// TIA Portal V18 export
FUNCTION "FC_Teach_Recipe_Transfer" : Void   // FC4, SCL
{ S7_Optimized_Access := 'TRUE' }
// stored: SetENOAutomatically false
   VAR_IN_OUT
      recipeIndex : USInt;
   END_VAR
BEGIN

   // Clamp recipe index to array bounds [1..10].
   // 
   IF #recipeIndex< 1 THEN
     #recipeIndex := 1;
   ELSIF #recipeIndex> 10 THEN
     #recipeIndex := 10;
   END_IF;

   // Block read/save if teach mode is not active.
   IF NOT "DB_PARAMETERS_TEACH".HMI_PAGE_CONTROL.TEACH_MODE_ACTIVE THEN
     "DB_PARAMETERS_TEACH".HMI_PAGE_CONTROL.READ_CHOOSED_RECIPE := FALSE;
     "DB_PARAMETERS_TEACH".HMI_PAGE_CONTROL.SAVE_CHANGES_IN_RECIPE := FALSE;
     RETURN;
   END_IF;

   // Read selected recipe into teach screen values.
   IF "DB_PARAMETERS_TEACH".HMI_PAGE_CONTROL.READ_CHOOSED_RECIPE THEN
     "DB_PARAMETERS_TEACH"."TEACH SCREEN VALUES" :=
     "DB_ALL_PROCESS_PARAMETERS".PRODUCT_TYPE[#recipeIndex];
    // "DB_ALL_PROCESS_PARAMETERS".ACTUAL_CHOOSEN_TYPE :=
   //  "DB_ALL_PROCESS_PARAMETERS".PRODUCT_TYPE[#recipeIndex];
     "DB_PARAMETERS_TEACH".HMI_PAGE_CONTROL.READ_CHOOSED_RECIPE := FALSE;
   END_IF;

   // Save teach screen values back into selected recipe.
    IF "DB_PARAMETERS_TEACH".HMI_PAGE_CONTROL.SAVE_CHANGES_IN_RECIPE THEN
     "DB_ALL_PROCESS_PARAMETERS".PRODUCT_TYPE[#recipeIndex] :=
     "DB_PARAMETERS_TEACH"."TEACH SCREEN VALUES";
    // "DB_ALL_PROCESS_PARAMETERS".ACTUAL_CHOOSEN_TYPE :=
   //  "DB_PARAMETERS_TEACH"."TEACH SCREEN VALUES";
     "DB_PARAMETERS_TEACH".HMI_PAGE_CONTROL.SAVE_CHANGES_IN_RECIPE := FALSE;
   END_IF;
END_FUNCTION
